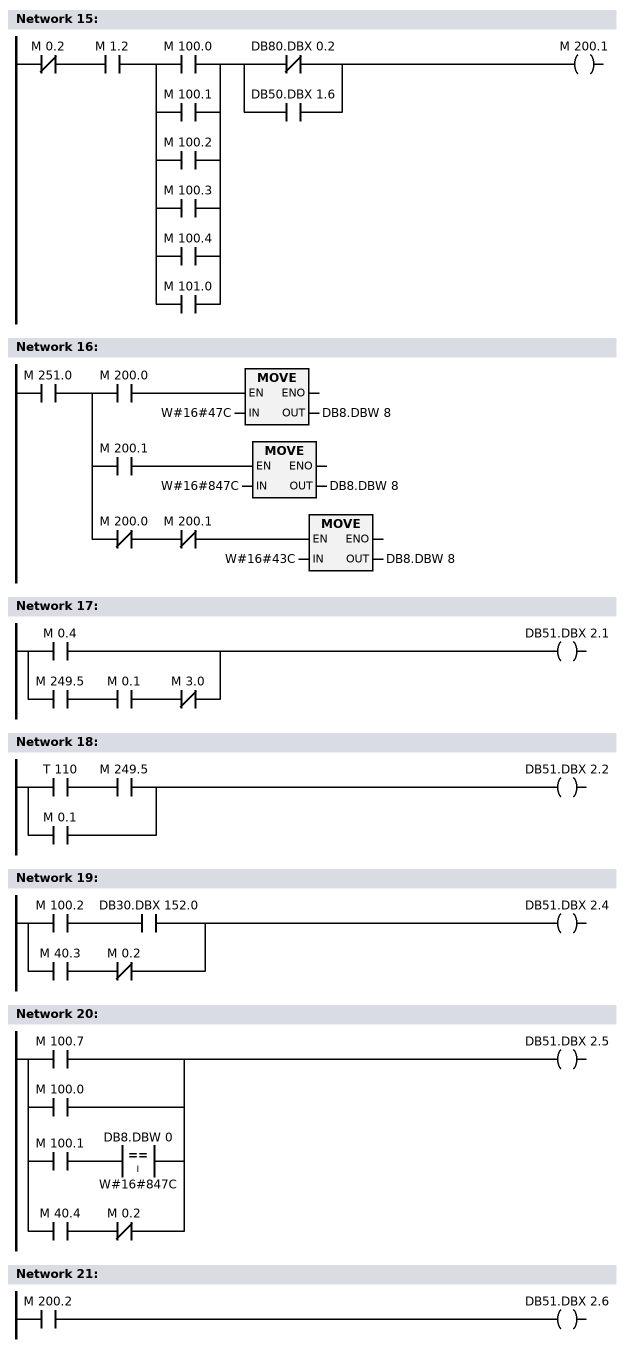
NETWORK
TITLE =
      AN    M 0.2;
      A     M 1.2;
      A(;
      O     M 100.0;
      O     M 100.1;
      O     M 100.2;
      O     M 100.3;
      O     M 100.4;
      O     M 101.0;
      );
      A(;
      ON    DB80.DBX 0.2;
      O     DB50.DBX 1.6;
      );
      =     M 200.1;
NETWORK
TITLE =
      A     M 251.0;
      =     L 0.0;
      A     L 0.0;
      A     M 200.0;
      JNB   M003;
      L     W#16#47C;
      T     DB8.DBW 8;
M003: NOP   0;
      A     L 0.0;
      A     M 200.1;
      JNB   M004;
      L     W#16#847C;
      T     DB8.DBW 8;
M004: NOP   0;
      A     L 0.0;
      AN    M 200.0;
      AN    M 200.1;
      JNB   M005;
      L     W#16#43C;
      T     DB8.DBW 8;
M005: NOP   0;
NETWORK
TITLE =
      O     M 0.4;
      O;
      A     M 249.5;
      A     M 0.1;
      AN    M 3.0;
      =     DB51.DBX 2.1;
NETWORK
TITLE =
      A     T 110;
      A     M 249.5;
      O     M 0.1;
      =     DB51.DBX 2.2;
NETWORK
TITLE =
      A     M 100.2;
      A     DB30.DBX 152.0;
      O;
      A     M 40.3;
      AN    M 0.2;
      =     DB51.DBX 2.4;
NETWORK
TITLE =
      O     M 100.7;
      O     M 100.0;
      O;
      A     M 100.1;
      A(;
      L     DB8.DBW 0;
      L     W#16#847C;
      ==I;
      );
      O;
      A     M 40.4;
      AN    M 0.2;
      =     DB51.DBX 2.5;
NETWORK
TITLE =
      A     M 200.2;
      =     DB51.DBX 2.6;
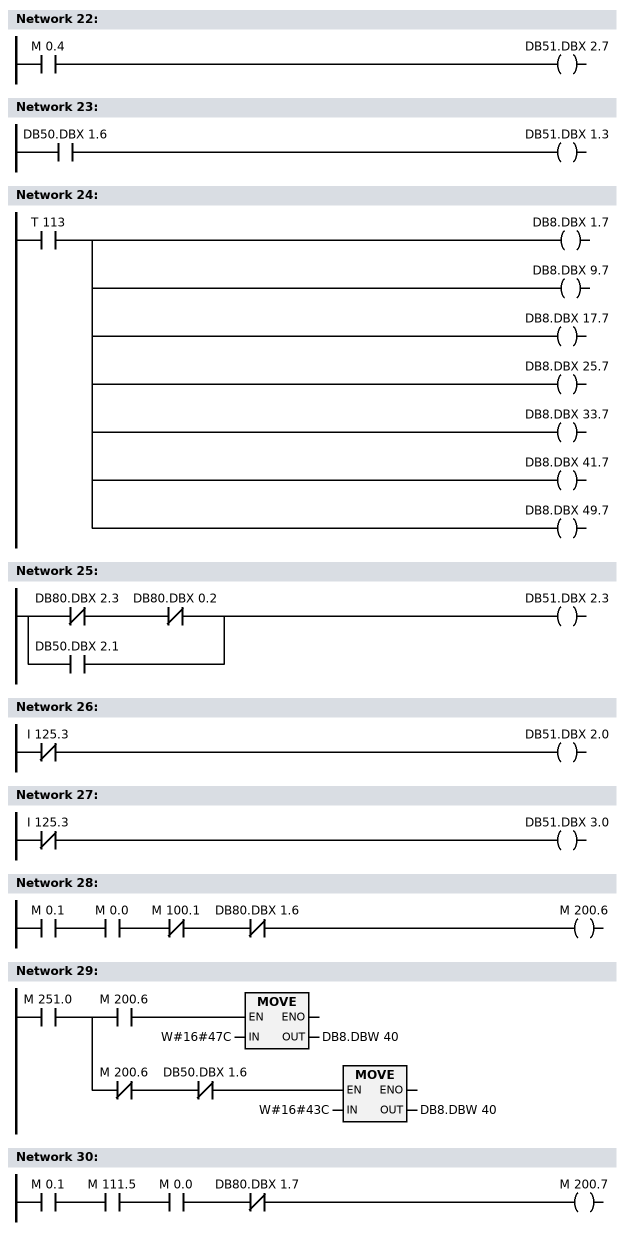
NETWORK
TITLE =
      A     M 0.4;
      =     DB51.DBX 2.7;
NETWORK
TITLE =
      A     DB50.DBX 1.6;
      =     DB51.DBX 1.3;
NETWORK
TITLE =
      A     T 113;
      =     DB8.DBX 1.7;
      =     DB8.DBX 9.7;
      =     DB8.DBX 17.7;
      =     DB8.DBX 25.7;
      =     DB8.DBX 33.7;
      =     DB8.DBX 41.7;
      =     DB8.DBX 49.7;
NETWORK
TITLE =
      AN    DB80.DBX 2.3;
      AN    DB80.DBX 0.2;
      O     DB50.DBX 2.1;
      =     DB51.DBX 2.3;
NETWORK
TITLE =
      AN    I 125.3;
      =     DB51.DBX 2.0;
NETWORK
TITLE =
      AN    I 125.3;
      =     DB51.DBX 3.0;
NETWORK
TITLE =
      A     M 0.1;
      A     M 0.0;
      AN    M 100.1;
      AN    DB80.DBX 1.6;
      =     M 200.6;
NETWORK
TITLE =
      A     M 251.0;
      =     L 0.0;
      A     L 0.0;
      A     M 200.6;
      JNB   M006;
      L     W#16#47C;
      T     DB8.DBW 40;
M006: NOP   0;
      A     L 0.0;
      AN    M 200.6;
      AN    DB50.DBX 1.6;
      JNB   M007;
      L     W#16#43C;
      T     DB8.DBW 40;
M007: NOP   0;
NETWORK
TITLE =
      A     M 0.1;
      A     M 111.5;
      A     M 0.0;
      AN    DB80.DBX 1.7;
      =     M 200.7;
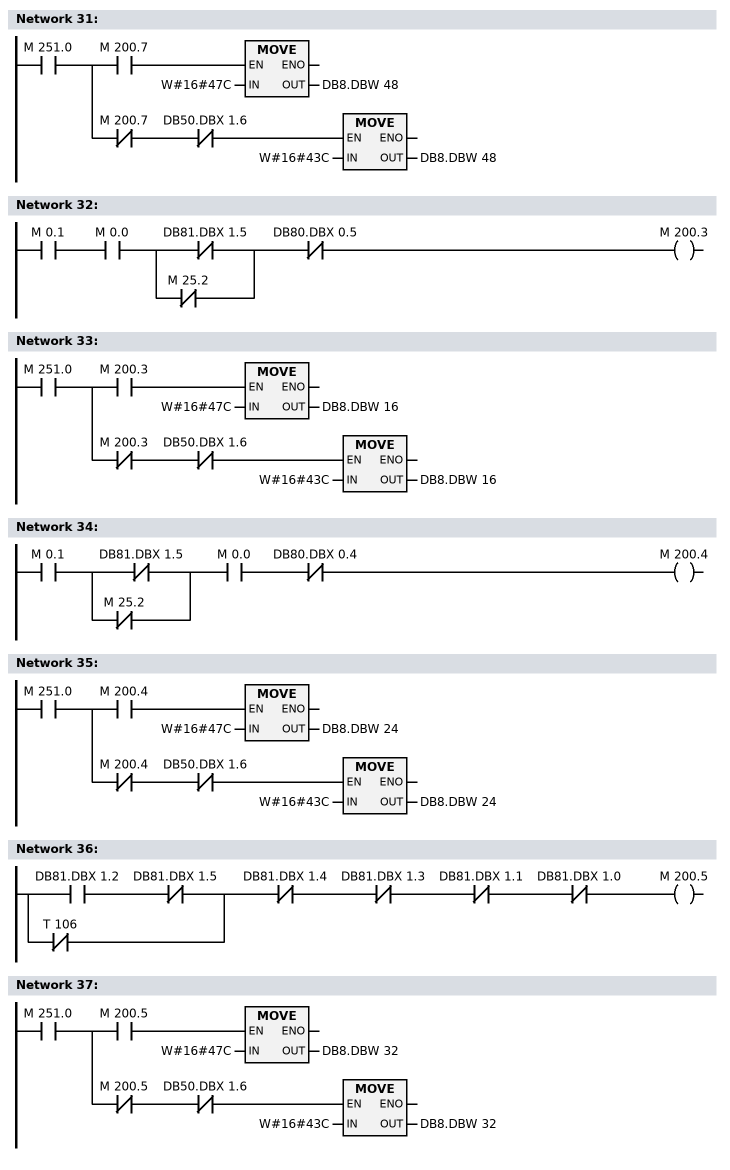
NETWORK
TITLE =
      A     M 251.0;
      =     L 0.0;
      A     L 0.0;
      A     M 200.7;
      JNB   M008;
      L     W#16#47C;
      T     DB8.DBW 48;
M008: NOP   0;
      A     L 0.0;
      AN    M 200.7;
      AN    DB50.DBX 1.6;
      JNB   M009;
      L     W#16#43C;
      T     DB8.DBW 48;
M009: NOP   0;
NETWORK
TITLE =
      A     M 0.1;
      A     M 0.0;
      A(;
      ON    DB81.DBX 1.5;
      ON    M 25.2;
      );
      AN    DB80.DBX 0.5;
      =     M 200.3;
NETWORK
TITLE =
      A     M 251.0;
      =     L 0.0;
      A     L 0.0;
      A     M 200.3;
      JNB   M010;
      L     W#16#47C;
      T     DB8.DBW 16;
M010: NOP   0;
      A     L 0.0;
      AN    M 200.3;
      AN    DB50.DBX 1.6;
      JNB   M011;
      L     W#16#43C;
      T     DB8.DBW 16;
M011: NOP   0;
NETWORK
TITLE =
      A     M 0.1;
      A(;
      ON    DB81.DBX 1.5;
      ON    M 25.2;
      );
      A     M 0.0;
      AN    DB80.DBX 0.4;
      =     M 200.4;
NETWORK
TITLE =
      A     M 251.0;
      =     L 0.0;
      A     L 0.0;
      A     M 200.4;
      JNB   M012;
      L     W#16#47C;
      T     DB8.DBW 24;
M012: NOP   0;
      A     L 0.0;
      AN    M 200.4;
      AN    DB50.DBX 1.6;
      JNB   M013;
      L     W#16#43C;
      T     DB8.DBW 24;
M013: NOP   0;
NETWORK
TITLE =
      A(;
      A     DB81.DBX 1.2;
      AN    DB81.DBX 1.5;
      ON    T 106;
      );
      AN    DB81.DBX 1.4;
      AN    DB81.DBX 1.3;
      AN    DB81.DBX 1.1;
      AN    DB81.DBX 1.0;
      =     M 200.5;
NETWORK
TITLE =
      A     M 251.0;
      =     L 0.0;
      A     L 0.0;
      A     M 200.5;
      JNB   M014;
      L     W#16#47C;
      T     DB8.DBW 32;
M014: NOP   0;
      A     L 0.0;
      AN    M 200.5;
      AN    DB50.DBX 1.6;
      JNB   M015;
      L     W#16#43C;
      T     DB8.DBW 32;
M015: NOP   0;
END_FUNCTION

FUNCTION FC 80 : VOID
VERSION : 0.1
BEGIN
// (block stored without names or comments; labels and parameter names are numbered)
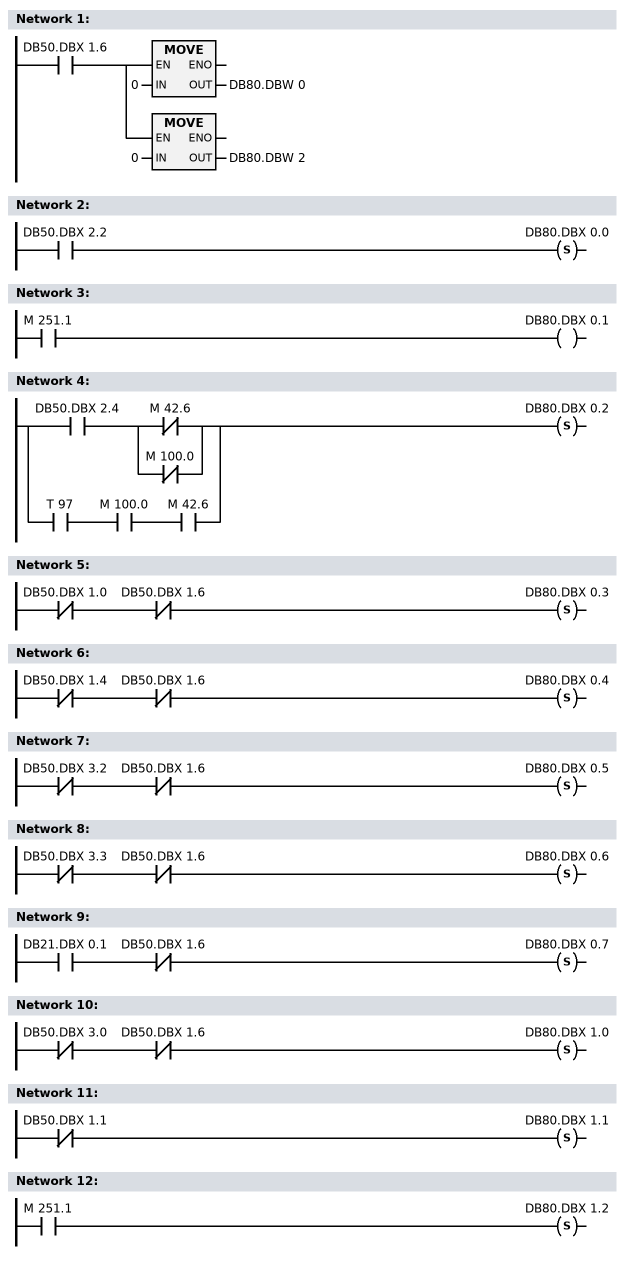
NETWORK
TITLE =
      A     DB50.DBX 1.6;
      =     L 0.0;
      A     L 0.0;
      JNB   M001;
      L     0;
      T     DB80.DBW 0;
M001: NOP   0;
      A     L 0.0;
      JNB   M002;
      L     0;
      T     DB80.DBW 2;
M002: NOP   0;
NETWORK
TITLE =
      A     DB50.DBX 2.2;
      S     DB80.DBX 0.0;
NETWORK
TITLE =
      A     M 251.1;
      =     DB80.DBX 0.1;
NETWORK
TITLE =
      A     DB50.DBX 2.4;
      A(;
      ON    M 42.6;
      ON    M 100.0;
      );
      O;
      A     T 97;
      A     M 100.0;
      A     M 42.6;
      S     DB80.DBX 0.2;
NETWORK
TITLE =
      AN    DB50.DBX 1.0;
      AN    DB50.DBX 1.6;
      S     DB80.DBX 0.3;
NETWORK
TITLE =
      AN    DB50.DBX 1.4;
      AN    DB50.DBX 1.6;
      S     DB80.DBX 0.4;
NETWORK
TITLE =
      AN    DB50.DBX 3.2;
      AN    DB50.DBX 1.6;
      S     DB80.DBX 0.5;
NETWORK
TITLE =
      AN    DB50.DBX 3.3;
      AN    DB50.DBX 1.6;
      S     DB80.DBX 0.6;
NETWORK
TITLE =
      A     DB21.DBX 0.1;
      AN    DB50.DBX 1.6;
      S     DB80.DBX 0.7;
NETWORK
TITLE =
      AN    DB50.DBX 3.0;
      AN    DB50.DBX 1.6;
      S     DB80.DBX 1.0;
NETWORK
TITLE =
      AN    DB50.DBX 1.1;
      S     DB80.DBX 1.1;
NETWORK
TITLE =
      A     M 251.1;
      S     DB80.DBX 1.2;
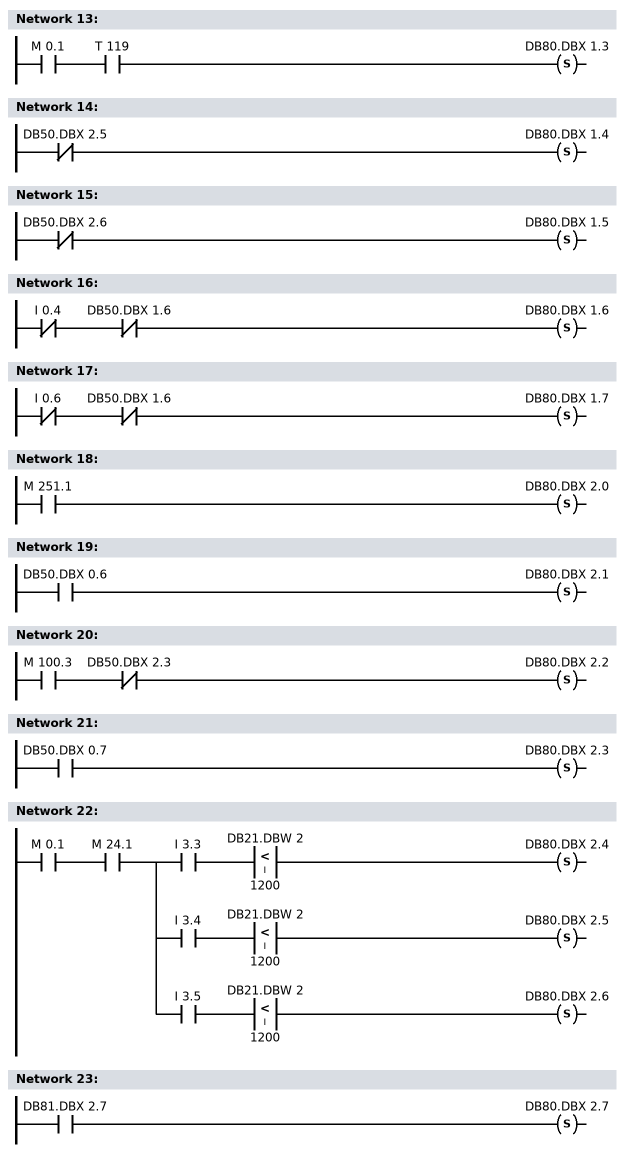
NETWORK
TITLE =
      A     M 0.1;
      A     T 119;
      S     DB80.DBX 1.3;
NETWORK
TITLE =
      AN    DB50.DBX 2.5;
      S     DB80.DBX 1.4;
NETWORK
TITLE =
      AN    DB50.DBX 2.6;
      S     DB80.DBX 1.5;
NETWORK
TITLE =
      AN    I 0.4;
      AN    DB50.DBX 1.6;
      S     DB80.DBX 1.6;
NETWORK
TITLE =
      AN    I 0.6;
      AN    DB50.DBX 1.6;
      S     DB80.DBX 1.7;
NETWORK
TITLE =
      A     M 251.1;
      S     DB80.DBX 2.0;
NETWORK
TITLE =
      A     DB50.DBX 0.6;
      S     DB80.DBX 2.1;
NETWORK
TITLE =
      A     M 100.3;
      AN    DB50.DBX 2.3;
      S     DB80.DBX 2.2;
NETWORK
TITLE =
      A     DB50.DBX 0.7;
      S     DB80.DBX 2.3;
NETWORK
TITLE =
      A     M 0.1;
      A     M 24.1;
      =     L 0.0;
      A     L 0.0;
      A     I 3.3;
      A(;
      L     DB21.DBW 2;
      L     1200;
      <I;
      );
      S     DB80.DBX 2.4;
      A     L 0.0;
      A     I 3.4;
      A(;
      L     DB21.DBW 2;
      L     1200;
      <I;
      );
      S     DB80.DBX 2.5;
      A     L 0.0;
      A     I 3.5;
      A(;
      L     DB21.DBW 2;
      L     1200;
      <I;
      );
      S     DB80.DBX 2.6;
NETWORK
TITLE =
      A     DB81.DBX 2.7;
      S     DB80.DBX 2.7;
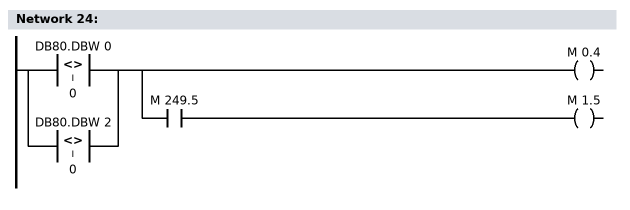
NETWORK
TITLE =
      O(;
      L     DB80.DBW 0;
      L     0;
      <>I;
      );
      O(;
      L     DB80.DBW 2;
      L     0;
      <>I;
      );
      =     L 0.0;
      A     L 0.0;
      BLD   102;
      =     M 0.4;
      A     L 0.0;
      A     M 249.5;
      =     M 1.5;
END_FUNCTION

FUNCTION FC 81 : VOID
VERSION : 0.1
BEGIN
// (block stored without names or comments; labels and parameter names are numbered)
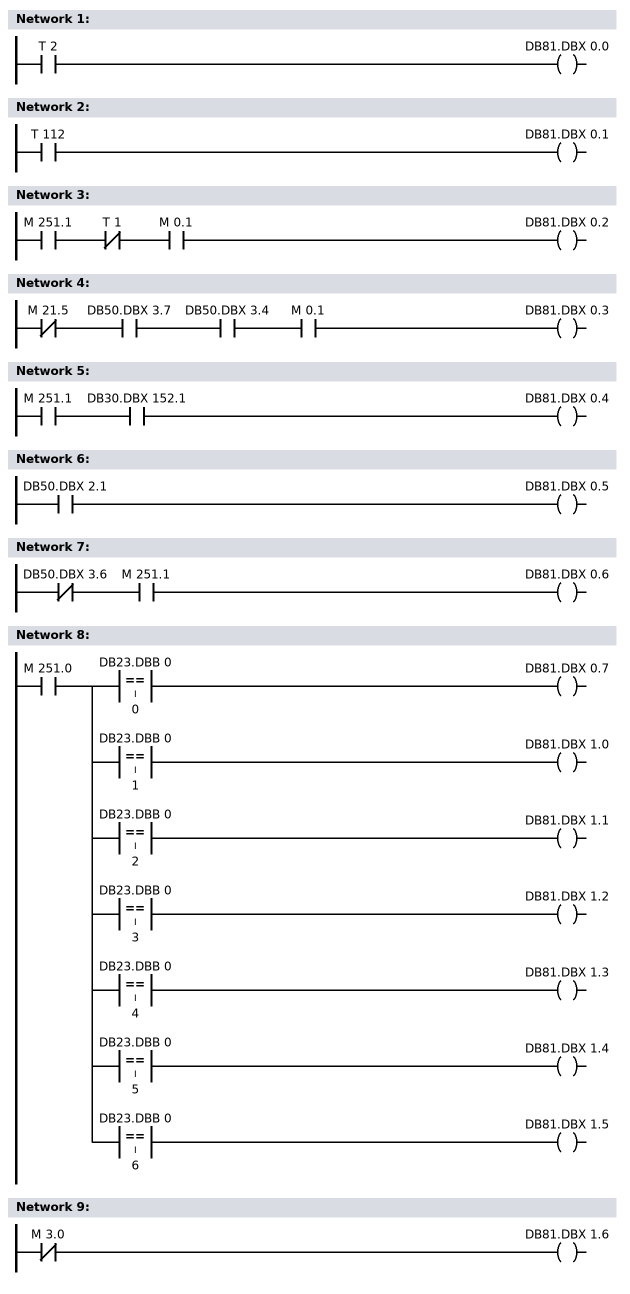
NETWORK
TITLE =
      A     T 2;
      =     DB81.DBX 0.0;
NETWORK
TITLE =
      A     T 112;
      =     DB81.DBX 0.1;
NETWORK
TITLE =
      A     M 251.1;
      AN    T 1;
      A     M 0.1;
      =     DB81.DBX 0.2;
NETWORK
TITLE =
      AN    M 21.5;
      A     DB50.DBX 3.7;
      A     DB50.DBX 3.4;
      A     M 0.1;
      =     DB81.DBX 0.3;
NETWORK
TITLE =
      A     M 251.1;
      A     DB30.DBX 152.1;
      =     DB81.DBX 0.4;
NETWORK
TITLE =
      A     DB50.DBX 2.1;
      =     DB81.DBX 0.5;
NETWORK
TITLE =
      AN    DB50.DBX 3.6;
      A     M 251.1;
      =     DB81.DBX 0.6;
NETWORK
TITLE =
      A     M 251.0;
      =     L 0.0;
      A     L 0.0;
      A(;
      L     DB23.DBB 0;
      L     0;
      ==I;
      );
      =     DB81.DBX 0.7;
      A     L 0.0;
      A(;
      L     DB23.DBB 0;
      L     1;
      ==I;
      );
      =     DB81.DBX 1.0;
      A     L 0.0;
      A(;
      L     DB23.DBB 0;
      L     2;
      ==I;
      );
      =     DB81.DBX 1.1;
      A     L 0.0;
      A(;
      L     DB23.DBB 0;
      L     3;
      ==I;
      );
      =     DB81.DBX 1.2;
      A     L 0.0;
      A(;
      L     DB23.DBB 0;
      L     4;
      ==I;
      );
      =     DB81.DBX 1.3;
      A     L 0.0;
      A(;
      L     DB23.DBB 0;
      L     5;
      ==I;
      );
      =     DB81.DBX 1.4;
      A     L 0.0;
      A(;
      L     DB23.DBB 0;
      L     6;
      ==I;
      );
      =     DB81.DBX 1.5;
NETWORK
TITLE =
      AN    M 3.0;
      =     DB81.DBX 1.6;
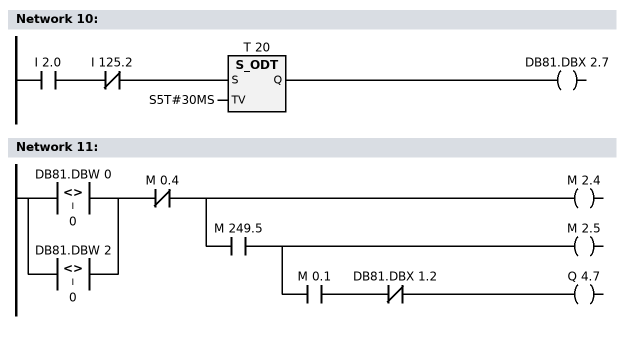
NETWORK
TITLE =
      A     I 2.0;
      AN    I 125.2;
      L     S5T#30MS;
      SD    T 20;
      NOP   0;
      NOP   0;
      NOP   0;
      A     T 20;
      =     DB81.DBX 2.7;
NETWORK
TITLE =
      A(;
      O(;
      L     DB81.DBW 0;
      L     0;
      <>I;
      );
      O(;
      L     DB81.DBW 2;
      L     0;
      <>I;
      );
      );
      AN    M 0.4;
      =     L 0.0;
      A     L 0.0;
      BLD   102;
      =     M 2.4;
      A     L 0.0;
      A     M 249.5;
      =     L 0.1;
      A     L 0.1;
      BLD   102;
      =     M 2.5;
      A     L 0.1;
      A     M 0.1;
      AN    DB81.DBX 1.2;
      =     Q 4.7;
END_FUNCTION

FUNCTION FC 103 : VOID
AUTHOR : GC
NAME : TRASFDB
VERSION : 0.0
BEGIN
// (block stored without names or comments; labels and parameter names are numbered)
NETWORK
TITLE =
      L     #PARAM2;
      T     LW 16;
      L     #PARAM5;
      T     LW 18;
      L     #PARAM1;
      T     LW 12;
      L     #PARAM4;
      T     LW 14;
M001: NOP   0;
      L     LW 16;
      SLW   4;
      T     LD 0;
      OPN   DB [LW 12];
      L     DBW [LD 0];
      T     LW 8;
      L     LW 18;
      SLW   4;
      T     LD 4;
      L     LW 8;
      OPN   DB [LW 14];
      T     DBW [LD 4];
      L     LW 16;
      L     1;
      +I;
      T     LW 16;
      L     LW 16;
      L     #PARAM3;
      >I;
      JC    M002;
      L     LW 18;
      L     1;
      +I;
      T     LW 18;
      JU    M001;
M002: NOP   0;
END_FUNCTION

DATA_BLOCK DB 1
VERSION : 0.1
BEGIN
// 106 bytes; values not shown
END_DATA_BLOCK

DATA_BLOCK DB 2
VERSION : 0.1
BEGIN
// 54 bytes; values not shown
END_DATA_BLOCK

DATA_BLOCK DB 3
VERSION : 0.1
BEGIN
// 102 bytes; values not shown
END_DATA_BLOCK

DATA_BLOCK DB 4
VERSION : 0.1
BEGIN
// 16 bytes; values not shown
END_DATA_BLOCK

DATA_BLOCK DB 7
VERSION : 0.1
UDT 7
BEGIN
END_DATA_BLOCK

DATA_BLOCK DB 8
VERSION : 0.1
UDT 8
BEGIN
END_DATA_BLOCK

DATA_BLOCK DB 18
VERSION : 0.1
BEGIN
// 102 bytes; values not shown
END_DATA_BLOCK

DATA_BLOCK DB 19
VERSION : 0.1
BEGIN
// 164 bytes; values not shown
END_DATA_BLOCK

DATA_BLOCK DB 20
AUTHOR : SIMATIC
FAMILY : TEC_FUNC
VERSION : 0.0
"COUNT"
BEGIN
END_DATA_BLOCK

DATA_BLOCK DB 21
VERSION : 0.1
UDT 1
BEGIN
END_DATA_BLOCK

DATA_BLOCK DB 22
VERSION : 0.1
UDT 2
BEGIN
END_DATA_BLOCK

DATA_BLOCK DB 23
VERSION : 0.1
UDT 1
BEGIN
END_DATA_BLOCK

DATA_BLOCK DB 24
VERSION : 0.1
UDT 2
BEGIN
END_DATA_BLOCK

DATA_BLOCK DB 30
VERSION : 0.0
FB 30
BEGIN
END_DATA_BLOCK

DATA_BLOCK DB 50
VERSION : 0.1
FB 50
BEGIN
END_DATA_BLOCK

DATA_BLOCK DB 51
VERSION : 0.1
FB 51
BEGIN
END_DATA_BLOCK

DATA_BLOCK DB 80
VERSION : 0.1
BEGIN
// 8 bytes; values not shown
END_DATA_BLOCK

DATA_BLOCK DB 81
VERSION : 0.1
BEGIN
// 8 bytes; values not shown
END_DATA_BLOCK

DATA_BLOCK DB 101
VERSION : 0.1
UDT 3
BEGIN
END_DATA_BLOCK

DATA_BLOCK DB 102
VERSION : 0.1
UDT 3
BEGIN
END_DATA_BLOCK

DATA_BLOCK DB 103
VERSION : 0.1
UDT 3
BEGIN
END_DATA_BLOCK

DATA_BLOCK DB 104
VERSION : 0.1
UDT 3
BEGIN
END_DATA_BLOCK

DATA_BLOCK DB 105
VERSION : 0.1
UDT 3
BEGIN
END_DATA_BLOCK

DATA_BLOCK DB 106
VERSION : 0.1
UDT 3
BEGIN
END_DATA_BLOCK

DATA_BLOCK DB 107
VERSION : 0.1
UDT 3
BEGIN
END_DATA_BLOCK

DATA_BLOCK DB 108
VERSION : 0.1
UDT 3
BEGIN
END_DATA_BLOCK

DATA_BLOCK DB 109
VERSION : 0.1
UDT 3
BEGIN
END_DATA_BLOCK

DATA_BLOCK DB 110
VERSION : 0.1
UDT 3
BEGIN
END_DATA_BLOCK

DATA_BLOCK DB 111
VERSION : 0.1
UDT 3
BEGIN
END_DATA_BLOCK

DATA_BLOCK DB 112
VERSION : 0.1
UDT 3
BEGIN
END_DATA_BLOCK

DATA_BLOCK DB 113
VERSION : 0.1
UDT 3
BEGIN
END_DATA_BLOCK

DATA_BLOCK DB 114
VERSION : 0.1
UDT 3
BEGIN
END_DATA_BLOCK

DATA_BLOCK DB 115
VERSION : 0.1
UDT 3
BEGIN
END_DATA_BLOCK

DATA_BLOCK DB 116
VERSION : 0.1
UDT 3
BEGIN
END_DATA_BLOCK

DATA_BLOCK DB 117
VERSION : 0.1
UDT 3
BEGIN
END_DATA_BLOCK

DATA_BLOCK DB 118
VERSION : 0.1
UDT 3
BEGIN
END_DATA_BLOCK

DATA_BLOCK DB 119
VERSION : 0.1
UDT 3
BEGIN
END_DATA_BLOCK

DATA_BLOCK DB 120
VERSION : 0.1
UDT 3
BEGIN
END_DATA_BLOCK

DATA_BLOCK DB 121
VERSION : 0.1
UDT 3
BEGIN
END_DATA_BLOCK

DATA_BLOCK DB 222
VERSION : 0.1
UDT 2
BEGIN
END_DATA_BLOCK

ORGANIZATION_BLOCK OB 1
VERSION : 0.1
BEGIN
// (block stored without names or comments; labels and parameter names are numbered)
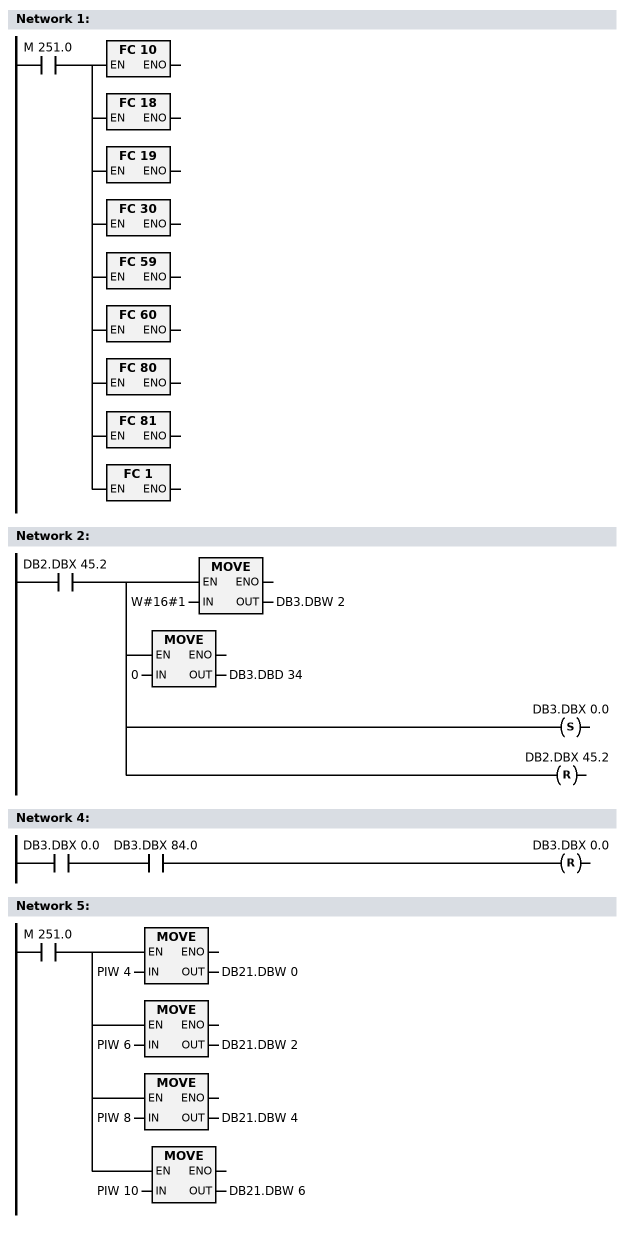
NETWORK
TITLE =
      A     M 251.0;
      =     L 20.0;
      A     L 20.0;
      JNB   M001;
      CALL  FC 10;
M001: NOP   0;
      A     L 20.0;
      JNB   M002;
      CALL  FC 18;
M002: NOP   0;
      A     L 20.0;
      JNB   M003;
      CALL  FC 19;
M003: NOP   0;
      A     L 20.0;
      JNB   M004;
      CALL  FC 30;
M004: NOP   0;
      A     L 20.0;
      JNB   M005;
      CALL  FC 59;
M005: NOP   0;
      A     L 20.0;
      JNB   M006;
      CALL  FC 60;
M006: NOP   0;
      A     L 20.0;
      JNB   M007;
      CALL  FC 80;
M007: NOP   0;
      A     L 20.0;
      JNB   M008;
      CALL  FC 81;
M008: NOP   0;
      A     L 20.0;
      JNB   M009;
      CALL  FC 1;
M009: NOP   0;
NETWORK
TITLE =
      A     DB2.DBX 45.2;
      =     L 20.0;
      A     L 20.0;
      JNB   M010;
      L     W#16#1;
      T     DB3.DBW 2;
M010: NOP   0;
      A     L 20.0;
      JNB   M011;
      L     0;
      T     DB3.DBD 34;
M011: NOP   0;
      A     L 20.0;
      BLD   102;
      S     DB3.DBX 0.0;
      A     L 20.0;
      BLD   102;
      R     DB2.DBX 45.2;
NETWORK
TITLE =
      A     M 251.0;
      =     L 20.0;
      BLD   103;
      A     DB3.DBX 0.0;
      =     L 20.3;
      BLD   103;
      BLD   9;
      =     L 25.0;
      CDB;
      OPN   DI 20;
      TAR2  LD 21;
      L     768;
      T     DIW 0;
      L     0;
      T     DIW 2;
      A     L 20.0;
      =     DIX 4.0;
      A     L 20.3;
      =     DIX 4.3;
      OPN   DI 3;
      L     DIW 2;
      OPN   DI 20;
      T     DIW 6;
      OPN   DI 3;
      L     DID 34;
      OPN   DI 20;
      T     DID 8;
      LAR2  P#DBX 0.0;
      UC    "COUNT";
      LAR2  LD 21;
      L     DID 14;
      OPN   DI 3;
      T     DID 86;
      OPN   DI 20;
      A     DIX 22.0;
      OPN   DI 3;
      =     DIX 84.0;
      OPN   DI 20;
      A     DIX 22.1;
      OPN   DI 3;
      =     DIX 66.0;
      OPN   DI 20;
      L     DIW 24;
      OPN   DI 3;
      T     DIW 68;
      OPN   DI 20;
      CDB;
      BLD   10;
      NOP   0;
NETWORK
TITLE =
      A     DB3.DBX 0.0;
      A     DB3.DBX 84.0;
      R     DB3.DBX 0.0;
NETWORK
TITLE =
      A     M 251.0;
      =     L 20.0;
      A     L 20.0;
      JNB   M012;
      L     PIW 4;
      T     DB21.DBW 0;
M012: NOP   0;
      A     L 20.0;
      JNB   M013;
      L     PIW 6;
      T     DB21.DBW 2;
M013: NOP   0;
      A     L 20.0;
      JNB   M014;
      L     PIW 8;
      T     DB21.DBW 4;
M014: NOP   0;
      A     L 20.0;
      JNB   M015;
      L     PIW 10;
      T     DB21.DBW 6;
M015: NOP   0;
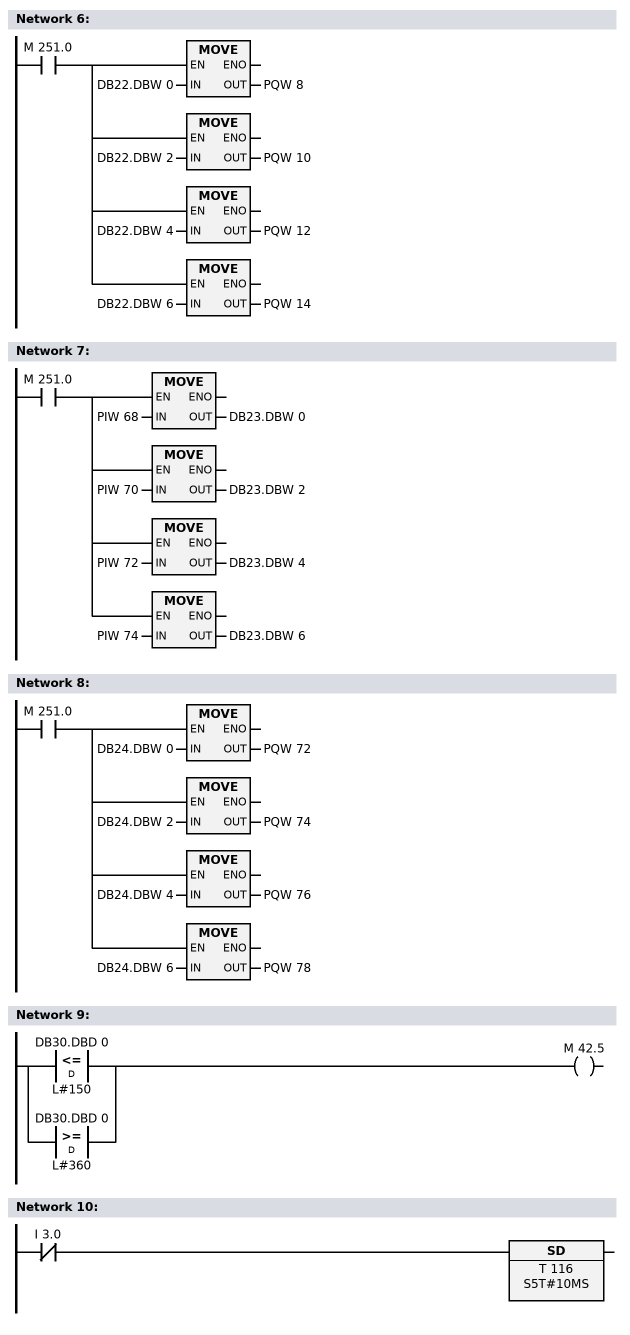
NETWORK
TITLE =
      A     M 251.0;
      =     L 20.0;
      A     L 20.0;
      JNB   M016;
      L     DB22.DBW 0;
      T     PQW 8;
M016: NOP   0;
      A     L 20.0;
      JNB   M017;
      L     DB22.DBW 2;
      T     PQW 10;
M017: NOP   0;
      A     L 20.0;
      JNB   M018;
      L     DB22.DBW 4;
      T     PQW 12;
M018: NOP   0;
      A     L 20.0;
      JNB   M019;
      L     DB22.DBW 6;
      T     PQW 14;
M019: NOP   0;
NETWORK
TITLE =
      A     M 251.0;
      =     L 20.0;
      A     L 20.0;
      JNB   M020;
      L     PIW 68;
      T     DB23.DBW 0;
M020: NOP   0;
      A     L 20.0;
      JNB   M021;
      L     PIW 70;
      T     DB23.DBW 2;
M021: NOP   0;
      A     L 20.0;
      JNB   M022;
      L     PIW 72;
      T     DB23.DBW 4;
M022: NOP   0;
      A     L 20.0;
      JNB   M023;
      L     PIW 74;
      T     DB23.DBW 6;
M023: NOP   0;
NETWORK
TITLE =
      A     M 251.0;
      =     L 20.0;
      A     L 20.0;
      JNB   M024;
      L     DB24.DBW 0;
      T     PQW 72;
M024: NOP   0;
      A     L 20.0;
      JNB   M025;
      L     DB24.DBW 2;
      T     PQW 74;
M025: NOP   0;
      A     L 20.0;
      JNB   M026;
      L     DB24.DBW 4;
      T     PQW 76;
M026: NOP   0;
      A     L 20.0;
      JNB   M027;
      L     DB24.DBW 6;
      T     PQW 78;
M027: NOP   0;
NETWORK
TITLE =
      O(;
      L     DB30.DBD 0;
      L     L#150;
      <=D;
      );
      O(;
      L     DB30.DBD 0;
      L     L#360;
      >=D;
      );
      =     M 42.5;
NETWORK
TITLE =
      AN    I 3.0;
      L     S5T#10MS;
      SD    T 116;
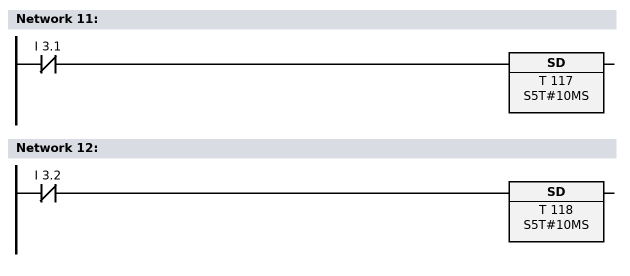
NETWORK
TITLE =
      AN    I 3.1;
      L     S5T#10MS;
      SD    T 117;
NETWORK
TITLE =
      AN    I 3.2;
      L     S5T#10MS;
      SD    T 118;
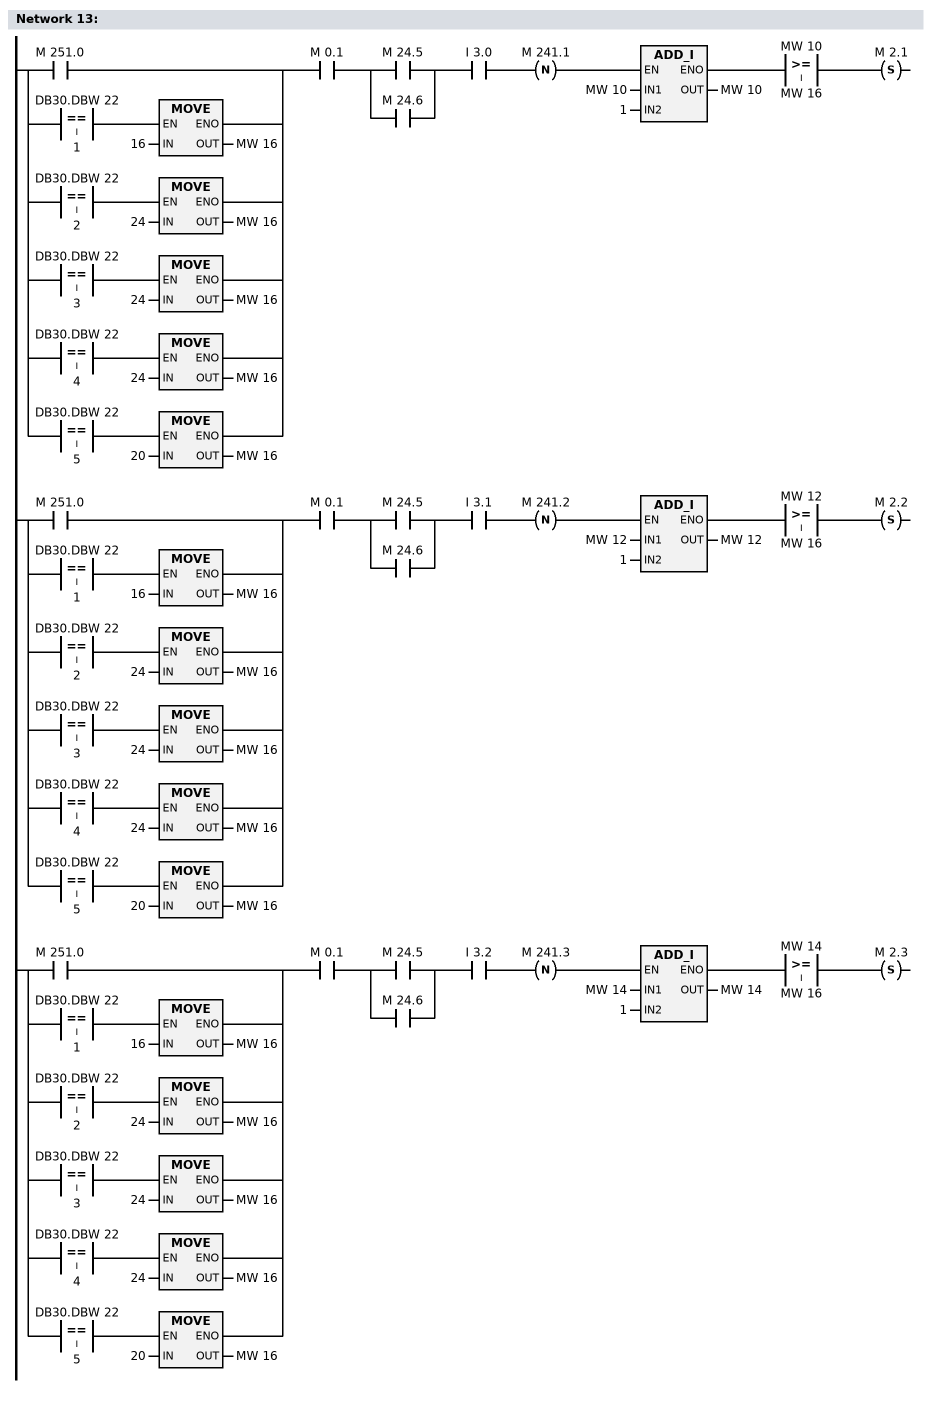
NETWORK
TITLE =
      A(;
      O     M 251.0;
      O(;
      A(;
      L     DB30.DBW 22;
      L     1;
      ==I;
      );
      JNB   M028;
      L     16;
      T     MW 16;
      SET;
      SAVE;
      CLR;
M028: A     BR;
      );
      O(;
      A(;
      L     DB30.DBW 22;
      L     2;
      ==I;
      );
      JNB   M029;
      L     24;
      T     MW 16;
      SET;
      SAVE;
      CLR;
M029: A     BR;
      );
      O(;
      A(;
      L     DB30.DBW 22;
      L     3;
      ==I;
      );
      JNB   M030;
      L     24;
      T     MW 16;
      SET;
      SAVE;
      CLR;
M030: A     BR;
      );
      O(;
      A(;
      L     DB30.DBW 22;
      L     4;
      ==I;
      );
      JNB   M031;
      L     24;
      T     MW 16;
      SET;
      SAVE;
      CLR;
M031: A     BR;
      );
      O(;
      A(;
      L     DB30.DBW 22;
      L     5;
      ==I;
      );
      JNB   M032;
      L     20;
      T     MW 16;
      SET;
      SAVE;
      CLR;
M032: A     BR;
      );
      );
      A     M 0.1;
      A(;
      O     M 24.5;
      O     M 24.6;
      );
      =     L 20.0;
      A(;
      A     L 20.0;
      A     I 3.0;
      FN    M 241.1;
      JNB   M033;
      L     MW 10;
      L     1;
      +I;
      T     MW 10;
      AN    OV;
      SAVE;
      CLR;
M033: A     BR;
      );
      A(;
      L     MW 10;
      L     MW 16;
      >=I;
      );
      S     M 2.1;
      A(;
      A     L 20.0;
      A     I 3.1;
      FN    M 241.2;
      JNB   M034;
      L     MW 12;
      L     1;
      +I;
      T     MW 12;
      AN    OV;
      SAVE;
      CLR;
M034: A     BR;
      );
      A(;
      L     MW 12;
      L     MW 16;
      >=I;
      );
      S     M 2.2;
      A(;
      A     L 20.0;
      A     I 3.2;
      FN    M 241.3;
      JNB   M035;
      L     MW 14;
      L     1;
      +I;
      T     MW 14;
      AN    OV;
      SAVE;
      CLR;
M035: A     BR;
      );
      A(;
      L     MW 14;
      L     MW 16;
      >=I;
      );
      S     M 2.3;
END_ORGANIZATION_BLOCK

ORGANIZATION_BLOCK OB 35
VERSION : 0.1
BEGIN
// (block stored without names or comments; labels and parameter names are numbered)
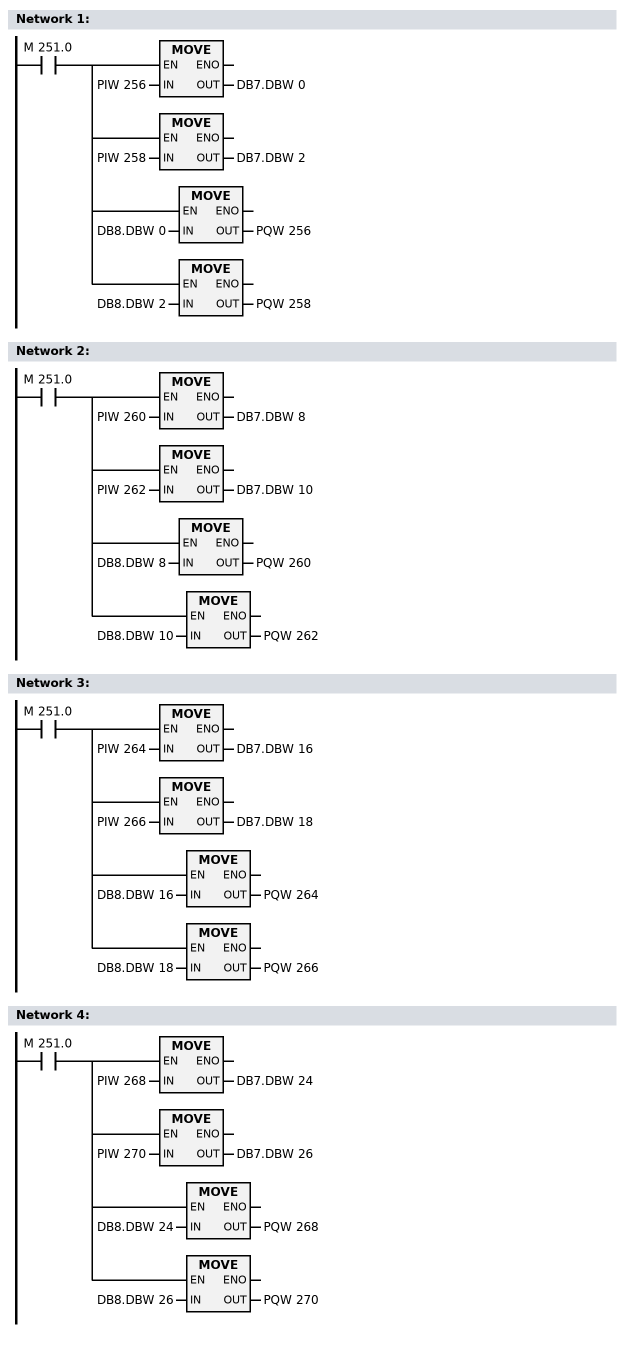
NETWORK
TITLE =
      A     M 251.0;
      =     L 20.0;
      A     L 20.0;
      JNB   M001;
      L     PIW 256;
      T     DB7.DBW 0;
M001: NOP   0;
      A     L 20.0;
      JNB   M002;
      L     PIW 258;
      T     DB7.DBW 2;
M002: NOP   0;
      A     L 20.0;
      JNB   M003;
      L     DB8.DBW 0;
      T     PQW 256;
M003: NOP   0;
      A     L 20.0;
      JNB   M004;
      L     DB8.DBW 2;
      T     PQW 258;
M004: NOP   0;
NETWORK
TITLE =
      A     M 251.0;
      =     L 20.0;
      A     L 20.0;
      JNB   M005;
      L     PIW 260;
      T     DB7.DBW 8;
M005: NOP   0;
      A     L 20.0;
      JNB   M006;
      L     PIW 262;
      T     DB7.DBW 10;
M006: NOP   0;
      A     L 20.0;
      JNB   M007;
      L     DB8.DBW 8;
      T     PQW 260;
M007: NOP   0;
      A     L 20.0;
      JNB   M008;
      L     DB8.DBW 10;
      T     PQW 262;
M008: NOP   0;
NETWORK
TITLE =
      A     M 251.0;
      =     L 20.0;
      A     L 20.0;
      JNB   M009;
      L     PIW 264;
      T     DB7.DBW 16;
M009: NOP   0;
      A     L 20.0;
      JNB   M010;
      L     PIW 266;
      T     DB7.DBW 18;
M010: NOP   0;
      A     L 20.0;
      JNB   M011;
      L     DB8.DBW 16;
      T     PQW 264;
M011: NOP   0;
      A     L 20.0;
      JNB   M012;
      L     DB8.DBW 18;
      T     PQW 266;
M012: NOP   0;
NETWORK
TITLE =
      A     M 251.0;
      =     L 20.0;
      A     L 20.0;
      JNB   M013;
      L     PIW 268;
      T     DB7.DBW 24;
M013: NOP   0;
      A     L 20.0;
      JNB   M014;
      L     PIW 270;
      T     DB7.DBW 26;
M014: NOP   0;
      A     L 20.0;
      JNB   M015;
      L     DB8.DBW 24;
      T     PQW 268;
M015: NOP   0;
      A     L 20.0;
      JNB   M016;
      L     DB8.DBW 26;
      T     PQW 270;
M016: NOP   0;
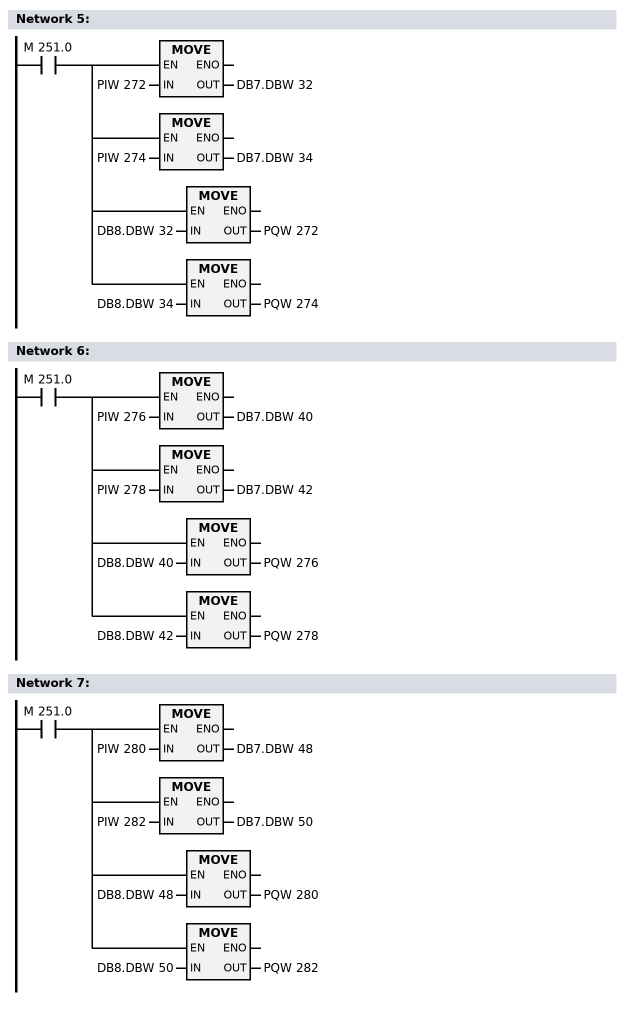
NETWORK
TITLE =
      A     M 251.0;
      =     L 20.0;
      A     L 20.0;
      JNB   M017;
      L     PIW 272;
      T     DB7.DBW 32;
M017: NOP   0;
      A     L 20.0;
      JNB   M018;
      L     PIW 274;
      T     DB7.DBW 34;
M018: NOP   0;
      A     L 20.0;
      JNB   M019;
      L     DB8.DBW 32;
      T     PQW 272;
M019: NOP   0;
      A     L 20.0;
      JNB   M020;
      L     DB8.DBW 34;
      T     PQW 274;
M020: NOP   0;
NETWORK
TITLE =
      A     M 251.0;
      =     L 20.0;
      A     L 20.0;
      JNB   M021;
      L     PIW 276;
      T     DB7.DBW 40;
M021: NOP   0;
      A     L 20.0;
      JNB   M022;
      L     PIW 278;
      T     DB7.DBW 42;
M022: NOP   0;
      A     L 20.0;
      JNB   M023;
      L     DB8.DBW 40;
      T     PQW 276;
M023: NOP   0;
      A     L 20.0;
      JNB   M024;
      L     DB8.DBW 42;
      T     PQW 278;
M024: NOP   0;
NETWORK
TITLE =
      A     M 251.0;
      =     L 20.0;
      A     L 20.0;
      JNB   M025;
      L     PIW 280;
      T     DB7.DBW 48;
M025: NOP   0;
      A     L 20.0;
      JNB   M026;
      L     PIW 282;
      T     DB7.DBW 50;
M026: NOP   0;
      A     L 20.0;
      JNB   M027;
      L     DB8.DBW 48;
      T     PQW 280;
M027: NOP   0;
      A     L 20.0;
      JNB   M028;
      L     DB8.DBW 50;
      T     PQW 282;
M028: NOP   0;
END_ORGANIZATION_BLOCK

ORGANIZATION_BLOCK OB 40
VERSION : 0.1
BEGIN
// (block stored without names or comments; labels and parameter names are numbered)
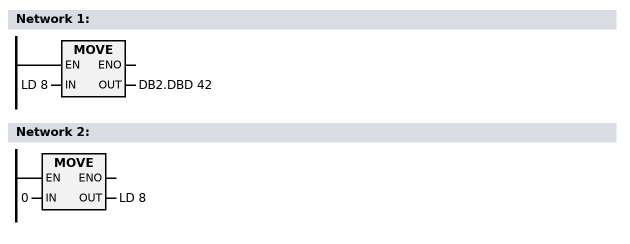
NETWORK
TITLE =
      L     LD 8;
      T     DB2.DBD 42;
NETWORK
TITLE =
      L     0;
      T     LD 8;
END_ORGANIZATION_BLOCK

ORGANIZATION_BLOCK OB 80
VERSION : 0.1
BEGIN
// (block stored without names or comments; labels and parameter names are numbered)
END_ORGANIZATION_BLOCK

ORGANIZATION_BLOCK OB 82
VERSION : 0.1
BEGIN
// (block stored without names or comments; labels and parameter names are numbered)
END_ORGANIZATION_BLOCK

ORGANIZATION_BLOCK OB 85
VERSION : 0.1
BEGIN
// (block stored without names or comments; labels and parameter names are numbered)
END_ORGANIZATION_BLOCK

ORGANIZATION_BLOCK OB 86
VERSION : 0.1
BEGIN
// (block stored without names or comments; labels and parameter names are numbered)
END_ORGANIZATION_BLOCK

ORGANIZATION_BLOCK OB 100
VERSION : 0.1
BEGIN
// (block stored without names or comments; labels and parameter names are numbered)
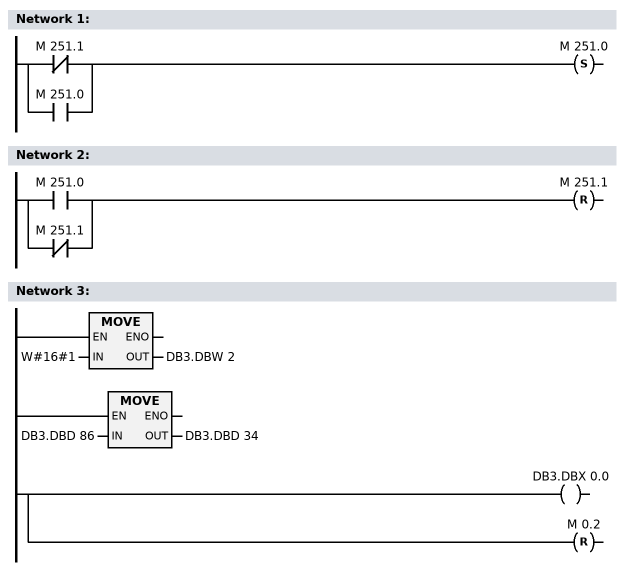
NETWORK
TITLE =
      ON    M 251.1;
      O     M 251.0;
      S     M 251.0;
NETWORK
TITLE =
      O     M 251.0;
      ON    M 251.1;
      R     M 251.1;
NETWORK
TITLE =
      L     W#16#1;
      T     DB3.DBW 2;
      L     DB3.DBD 86;
      T     DB3.DBD 34;
      SET;
      =     DB3.DBX 0.0;
      R     M 0.2;
END_ORGANIZATION_BLOCK

ORGANIZATION_BLOCK OB 121
VERSION : 0.1
BEGIN
// (block stored without names or comments; labels and parameter names are numbered)
END_ORGANIZATION_BLOCK

ORGANIZATION_BLOCK OB 122
VERSION : 0.1
BEGIN
// (block stored without names or comments; labels and parameter names are numbered)
END_ORGANIZATION_BLOCK
